FUNCTION_BLOCK FB_Factory

VAR
	fbTon : TON;
	fbTof : TOF;
	
	bMotorOn : BOOL;
	bFanOn : BOOL;
	
	tFanStartDelay : TIME := T#3S;
	tFanOffDelay : TIME := T#10s;
END_VAR


	fbTon(IN := bMotorOn, PT := tFanStartDelay);
	IF fbTon.Q THEN
		bFanOn := TRUE;
	END_IF
	fbTof(IN := bMotorOn , PT := tFanOffDelay);
	IF NOT fbTof.Q THEN
		bFanOn := FALSE;
	END_IF

END_FUNCTION_BLOCK

(* stored: Version 1.1.0.1, ProductVersion 3.1.4024.16
   POU FB_Factory: Id {ceceda62-7ae7-4377-8eaa-3edcee35a4c3}, SpecialFunc None *)
